Staubli VAL3: start.pgx

program start()
begin
  // clean the screen
  userPage()
  cls()
  // create the 2 task
  taskCreate "comunication",10,comunication()
  delay(0.1)
  taskCreate "check",10,check()
end
